{attribute 'linkalways'} 
{attribute 'no_explicit_call' := 'This FB is a CLASS and must be accessed using methods or properties'}
{attribute 'enable_dynamic_creation'}
FUNCTION_BLOCK Node_F_VN_ConvexHullPoints EXTENDS VisionNode
VAR
    ipPointSet : _ITcVnContainer;
    ipConvexHull : _ITcVnContainer;
    hrPrev : _HRESULT(S_OK);
	hresult : _HRESULT(S_OK);
END_VAR

METHOD PUBLIC  Clone : I_Node
VAR
	pNode : POINTER TO Node_F_VN_ConvexHullPoints;
END_VAR
pNode := __NEW(Node_F_VN_ConvexHullPoints);
Clone := pNode^;
END_METHOD

METHOD FB_init : BOOL
VAR_INPUT
	bInitRetains : BOOL; // if TRUE, the retain variables are initialized (warm start / cold start)
	bInCopyCode : BOOL;  // if TRUE, the instance afterwards gets moved into the copy code (online change)
END_VAR
AddInput('ipPointSet', ipPointSet);
AddInput('hrPrev', hrPrev);
AddOutput('ipConvexHull', ipConvexHull);
AddOutput('hresult',hresult);
END_METHOD

METHOD PROTECTED OnExecute
hresult.Value := F_VN_ConvexHullPoints(
	ipPointSet := ipPointSet.Value,
    ipConvexHull := ipConvexHull.Value,
	hrPrev:= hrPrev.Value);
END_METHOD

METHOD PUBLIC PreExecutionCheck
VAR_INPUT
	Check : I_PreExecutionChecks;
END_VAR
Check.IsTrue(ipPointSet.IsValid, 'ipPointSet must be a valid container');
Check.IsTrue((ipPointSet.IsType(TC_GLOBAL_CONST_LIST.ContainerType_Vector_TcVnPoint2_DINT) OR
              ipPointSet.IsType(TC_GLOBAL_CONST_LIST.ContainerType_Vector_TcVnPoint2_REAL)),
              'ipPointSet contains incorrect type');
END_METHOD

END_FUNCTION_BLOCK

(* stored: Version 1.1.0.1, ProductVersion 3.1.4026.13
   POU Node_F_VN_ConvexHullPoints: Id {51293896-4d4b-07a3-1128-f305c39d480f}, SpecialFunc None
   Folder Constructor: Id {050fc972-808c-087c-2e10-e6b0c587690b}
   Method Clone: Id {e596c0aa-e6a9-0f2f-2f84-b5d2914d7665}
   Method FB_init: Id {abe8c629-07ea-03f3-0276-b87b69b416d2}
   Method OnExecute: Id {09be0611-ea9f-01ef-2325-2414aecc6912}
   Method PreExecutionCheck: Id {80d69589-41a6-03f9-0af2-f10093cccaae} *)
